FUNCTION_BLOCK sequence_E_04_AX (* Sequence with 4 Outputs, Transition by EVENT, with AX Adapter *)
  (* Standard: 61499-2; Description: Copyright (c) 2024 HR Agrartechnik GmbH This program and the accompanying materials are made available under the terms of the Eclipse Public License 2.0 which is available at https://www.eclipse.org/legal/epl-2.0/ SPDX-License-Identifier: EPL-2.0 *)
  (* Version 1.0, 2024-03-02, Franz Höpfinger, HR Agrartechnik GmbH *)
  PACKAGE logiBUS::utils::sequence::event;
  IMPORT logiBUS::utils::sequence::const::sequence;
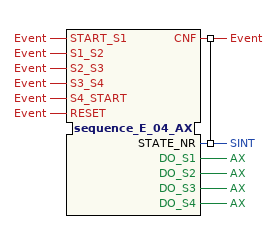
  EVENT_INPUT
    START_S1; (* jump from START to State_01 *)
    S1_S2; (* jump from State_01 to State_02 *)
    S2_S3; (* jump from State_02 to State_03 *)
    S3_S4; (* jump from State_03 to State_04 *)
    S4_START; (* jump from State_04 to START *)
    RESET; (* Reset from any State to START *)
  END_EVENT
  EVENT_OUTPUT
    CNF WITH STATE_NR; (* Execution Confirmation *)
  END_EVENT
  VAR_OUTPUT
    STATE_NR : SINT; (* State Number, START = 0, State_01 = 1 and so on. *)
  END_VAR
  PLUGS
    DO_S1 : adapter::types::unidirectional::AX; (* Output if State_01 is active *)
    DO_S2 : adapter::types::unidirectional::AX; (* Output if State_02 is active *)
    DO_S3 : adapter::types::unidirectional::AX; (* Output if State_03 is active *)
    DO_S4 : adapter::types::unidirectional::AX; (* Output if State_04 is active *)
  END_PLUGS
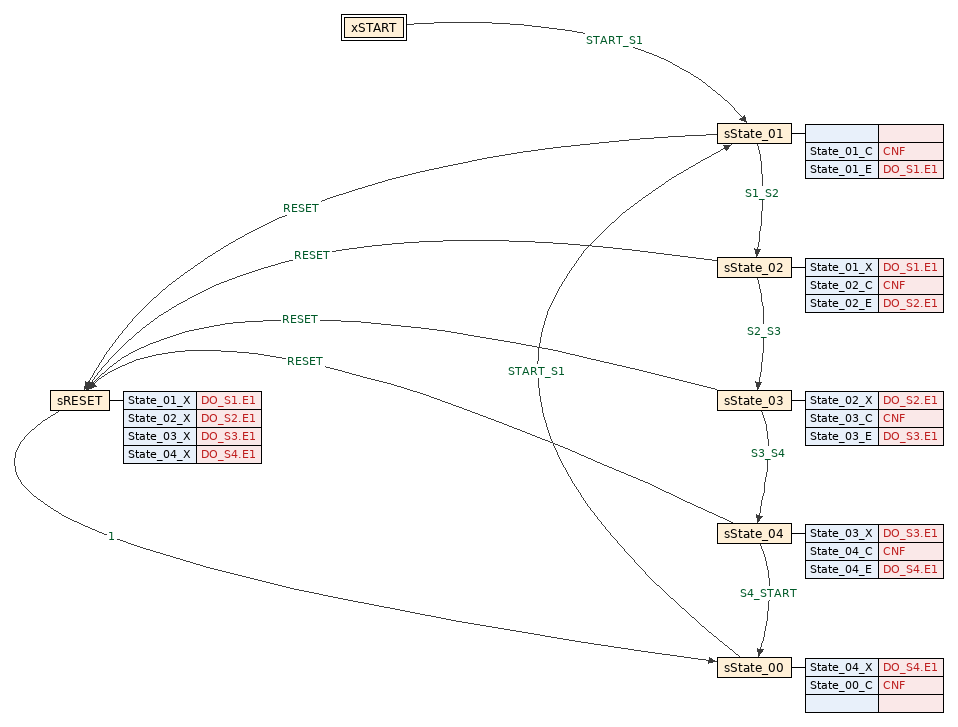
  EC_STATES
    xSTART; (* Initial State *)
    sState_01 : State_01_C -> CNF, State_01_E -> DO_S1.E1;
    sState_02 : State_01_X -> DO_S1.E1, State_02_C -> CNF, State_02_E -> DO_S2.E1;
    sState_03 : State_02_X -> DO_S2.E1, State_03_C -> CNF, State_03_E -> DO_S3.E1;
    sState_04 : State_03_X -> DO_S3.E1, State_04_C -> CNF, State_04_E -> DO_S4.E1;
    sState_00 : State_04_X -> DO_S4.E1, State_00_C -> CNF;
    sRESET : State_01_X -> DO_S1.E1, State_02_X -> DO_S2.E1, State_03_X -> DO_S3.E1, State_04_X -> DO_S4.E1;
  END_STATES
  EC_TRANSITIONS
    sState_01 TO sState_02 := S1_S2;
    sState_02 TO sState_03 := S2_S3;
    sState_03 TO sState_04 := S3_S4;
    sState_00 TO sState_01 := START_S1;
    sState_04 TO sState_00 := S4_START;
    xSTART TO sState_01 := START_S1;
    sState_01 TO sRESET := RESET;
    sState_04 TO sRESET := RESET;
    sState_02 TO sRESET := RESET;
    sState_03 TO sRESET := RESET;
    sRESET TO sState_00 := 1;
  END_TRANSITIONS
  ALGORITHM State_00_C IN ST:
 // State_00 Confirmation Step
STATE_NR := sequence::State_00;
  END_ALGORITHM
  ALGORITHM State_01_C IN ST:
 // State_01 Confirmation Step
STATE_NR := sequence::State_01;
  END_ALGORITHM
  ALGORITHM State_02_C IN ST:
 // State_02 Confirmation Step
STATE_NR := sequence::State_02;
  END_ALGORITHM
  ALGORITHM State_03_C IN ST:
 // State_03 Confirmation Step
STATE_NR := sequence::State_03;
  END_ALGORITHM
  ALGORITHM State_04_C IN ST:
 // State_04 Confirmation Step
STATE_NR := sequence::State_04;
  END_ALGORITHM
  ALGORITHM State_01_E IN ST:
 // State_01 Entry Step
DO_S1.D1 := BOOL#TRUE; // ON
  END_ALGORITHM
  ALGORITHM State_01_X IN ST:
 // State_01 Exit Step
DO_S1.D1 := BOOL#FALSE;
  END_ALGORITHM
  ALGORITHM State_02_E IN ST:
 // State_02 Entry Step
DO_S2.D1 := BOOL#TRUE; // ON
  END_ALGORITHM
  ALGORITHM State_02_X IN ST:
 // State_02 Exit Step
DO_S2.D1 := BOOL#FALSE;
  END_ALGORITHM
  ALGORITHM State_03_E IN ST:
 // State_03 Entry Step
DO_S3.D1 := BOOL#TRUE; // ON
  END_ALGORITHM
  ALGORITHM State_03_X IN ST:
 // State_03 Exit Step
DO_S3.D1 := BOOL#FALSE;
  END_ALGORITHM
  ALGORITHM State_04_E IN ST:
 // State_04 Entry Step
DO_S4.D1 := BOOL#TRUE; // ON
  END_ALGORITHM
  ALGORITHM State_04_X IN ST:
 // State_04 Exit Step
DO_S4.D1 := BOOL#FALSE;
  END_ALGORITHM
END_FUNCTION_BLOCK
